PROGRAM MAIN
VAR
END_VAR

END_PROGRAM

(* stored: Version 1.1.0.1
   POU MAIN: Id {98200c5f-463b-4f36-8ea6-4cbeafb39194} *)
